FUNCTION_BLOCK Grade_Comandos_HMI (* Service Interface Function Block Type *)
  (* Standard: 61499-2 *)
  (* Version 0.0, 2/24/2026, template *)
  PACKAGE Hidryco.HidrycoLib;
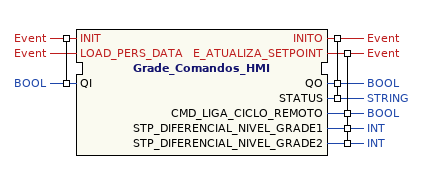
  EVENT_INPUT
    INIT WITH QI;
    LOAD_PERS_DATA;
  END_EVENT
  EVENT_OUTPUT
    INITO WITH QO, STATUS;
    E_ATUALIZA_SETPOINT WITH CMD_LIGA_CICLO_REMOTO, STP_DIFERENCIAL_NIVEL_GRADE1, STP_DIFERENCIAL_NIVEL_GRADE2;
  END_EVENT
  VAR_INPUT
    QI : BOOL;
  END_VAR
  VAR_OUTPUT
    QO : BOOL; (* Event Output Qualifier *)
    STATUS : STRING; (* Service Status *)
    CMD_LIGA_CICLO_REMOTO : BOOL; (* 1 - Liga Ciclo Remoto, 0 - Desliga Ciclo Remoto *)
    STP_DIFERENCIAL_NIVEL_GRADE1 : INT; (* Valor escalonado, ex: 0.0-100.0% = 0-1000 *)
    STP_DIFERENCIAL_NIVEL_GRADE2 : INT; (* Valor escalonado, ex: 0.0-100.0% = 0-1000 *)
  END_VAR
  SERVICE /
    SEQUENCE 
    END_SEQUENCE
  END_SERVICE
END_FUNCTION_BLOCK
